INTERFACE PUBLIC ResettingCommands

METHOD PUBLIC Abort
END_METHOD

METHOD PUBLIC StateComplete
END_METHOD

METHOD PUBLIC Stop
END_METHOD

END_INTERFACE

(* stored: Version 1.1.0.1, ProductVersion 3.1.4026.12
   Itf ResettingCommands: Id {8d330c53-dd73-014c-3c2b-ac3d4e386b6d}
   Method Abort: Id {1a8fcfa0-7e85-4966-8174-eeac0f03734a}
   Method StateComplete: Id {e2b64fcf-c81a-4a11-9ec4-2b60462de974}
   Method Stop: Id {f4b6d894-ef87-49b2-b8df-669443a04d76} *)
